(* CoDeSys 2.3.9.48 project: PLC_JBI.pro *)
(* Libraries: Util.lib 18.5.10 17:14:28, STANDARD.LIB 4.10.05 13:14:46, IECSFC.LIB 13.4.06 17:51:28, SYSLIBTIME.LIB 20.2.06 15:31:16, SYSTASKINFO.LIB 20.2.06 15:31:38, ANALYZATION.LIB 5.10.99 11:05:06, SYSLIBCALLBACK.LIB 20.2.06 15:31:08 *)

(* PLC configuration (modules and I/O channels)
Fast Counters [OWEN_ID531] node 0, in %IB0 out %QB0 {Visibility = No}
  di1_water AT %IW0.0 [WordInput] Fast counter 1
  di2_plast AT %IW0.1 [WordInput] Fast counter 2
AT %IB1.0 [ByteInput] 8 discrete inputs
AT %IB1.1 [ByteInput] 8 discrete inputs
Fast discrete outputs [OWEN_ID570] node 2, in %IB2 out %QB2 {SafeValueBool = FALSE; SafeValueBool = FALSE; SafeValueBool = FALSE; SafeValueBool = FALSE; Visibility = No}
  do1_comp_1 AT %QX2.0 [BitOutput] Fast discrete output 1
  do2_comp_2 AT %QX2.1 [BitOutput] Fast discrete output 2
  do3_comp_3 AT %QX2.2 [BitOutput] Fast discrete output 3
  do4_sem_raz AT %QX2.3 [BitOutput] Fast discrete output 4
Discrete outputs - 8 [ID131] node 3, in %IB3 out %QB3 {SafeValueByte = 0; Visibility = No; PinCount = 10}
  AT %QB3.0 [ByteOutput] 8 discrete outputs
Special input [ID103] node 4, in %IB4 out %QB4 {Filtrationtime = 1000; PinCount = 1; WatchDogPeriod = 400; PollPeriod = 3000; Visibility = No}
  AT %IX4.0 [BitInput] Special input
Special output [ID104] node 5, in %IB5 out %QB5 {Visibility = No; PinCount = 1}
  AT %QX5.0 [BitOutput] Special output
DCON (Master) [DCON_MASTER_ID452] node 6, in %IB6 out %QB6 {Visibility = No}
  AT %QW6.0 [WordOutput] Last error
  RS-485-2 [COM3_USART] node 0, in %IB6.0 out %QB6.0 {CommunicationSpeed = 11520; Parity = NO PARITY CHECK; BitLength = 8 bits; StopLength = One stop bit; InterfaceType = RS232; FrameOriented = ASCII; Timeout = 0; Visibility = No}
  Universal DCON device [ID2100] node 1, in %IB6.1 out %QB6.1 {ReqFormat = [15s]; GoodResponseFormat = !01[15s]; BadResponseFormat = ?; ServiceTimeout = 150; RequestType = By poll time; PeriodOfService = 100; Visibility = No}
    AT %QW6.1.0 [WordOutput] Status
cmd_plast AT %QB6.1.0.0 [StringOutput]
cntr_plast AT %IB6.1.1.0 [StringInput]
Universal DCON device [ID2100] node 2, in %IB6.2 out %QB6.2 {ReqFormat = [15s]; GoodResponseFormat = !02[15s]; BadResponseFormat = ?; ServiceTimeout = 150; RequestType = By poll time; PeriodOfService = 100; Visibility = No}
  AT %QW6.2.0 [WordOutput] Status
cmd_water AT %QB6.2.0.0 [StringOutput]
cntr_water AT %IB6.2.1.0 [StringInput]
Universal DCON device [ID2100] node 3, in %IB6.3 out %QB6.3 {ReqFormat = #01; GoodResponseFormat = >[8s]; BadResponseFormat = ?; ServiceTimeout = 150; RequestType = By poll time; PeriodOfService = 100; Visibility = No}
  AT %QW6.3.0 [WordOutput] Status
mVolt_sem AT %IB6.3.0.0 [StringInput]
Universal DCON device [ID2100] node 4, in %IB6.4 out %QB6.4 {ReqFormat = #02; GoodResponseFormat = >[8s]; BadResponseFormat = ?; ServiceTimeout = 150; RequestType = By poll time; PeriodOfService = 100; Visibility = No}
  AT %QW6.4.0 [WordOutput] Status
mVolt_sir AT %IB6.4.0.0 [StringInput]
AT %QW6.5.0 [WordOutput] Status
mVolt_wtr AT %IB6.5.0.0 [StringInput]
TCP [TCP_ID221] node 0, in %IB7.0.0 out %QB7.0.0 {RemotePort = 502; Visibility = No}
TCP [TCP_ID221] node 1, in %IB7.0.1 out %QB7.0.1 {RemotePort = 502; Visibility = No}
TCP [TCP_ID221] node 2, in %IB7.0.2 out %QB7.0.2 {RemotePort = 502; Visibility = No}
TCP [TCP_ID221] node 3, in %IB7.0.3 out %QB7.0.3 {RemotePort = 502; Visibility = No}
TCP [TCP_ID221] node 4, in %IB7.0.4 out %QB7.0.4 {RemotePort = 502; Visibility = No}
TCP [TCP_ID221] node 5, in %IB7.0.5 out %QB7.0.5 {RemotePort = 502; Visibility = No}
RS-232 [COM2_USART] node 6, in %IB7.0.6 out %QB7.0.6 {CommunicationSpeed = 11520; Parity = NO PARITY CHECK; BitLength = 8 bits; StopLength = One stop bit; InterfaceType = RS232; FrameOriented = RTU; Timeout = 10; Visibility = No}
Debug RS-232 [DEBUG_USART] node 7, in %IB7.0.7 out %QB7.0.7 {CommunicationSpeed = 11520; Parity = NO PARITY CHECK; BitLength = 8 bits; StopLength = One stop bit; InterfaceType = RS232; FrameOriented = RTU; Timeout = 10; Visibility = No}
8 bits [8Bit] node 1, in %IB7.1 out %QB7.1
  pc_mln_out1 AT %QB7.1.0 [ByteOutput] reg 0
8 bits [8Bit] node 2, in %IB7.2 out %QB7.2
  pc_mnl_out2 AT %QB7.2.0 [ByteOutput] reg 8
8 bits [8Bit] node 3, in %IB7.3 out %QB7.3
  pc_mnl_out3 AT %QB7.3.0 [ByteOutput] reg 16
8 bits [8Bit] node 4, in %IB7.4 out %QB7.4
  pc_mnl_in1 AT %QB7.4.0 [ByteOutput] reg 24
8 bits [8Bit] node 5, in %IB7.5 out %QB7.5
  pc_mnl_in2 AT %QB7.5.0 [ByteOutput] reg 32
8 bits [8Bit] node 6, in %IB7.6 out %QB7.6
  pc_mnl_in3 AT %QB7.6.0 [ByteOutput] reg 40
8 bits [8Bit] node 7, in %IB7.7 out %QB7.7
  AT %QB7.7.0 [ByteOutput] reg 48
8 bits [8Bit] node 8, in %IB7.8 out %QB7.8
  AT %QB7.8.0 [ByteOutput] reg 56
mb_local_sikl AT %QW7.9.0 [WordOutput]
mb_working_mode AT %QW7.10.0 [WordOutput]
mb_sikl AT %QW7.11.0 [WordOutput]
mb_tmr_conv AT %QW7.12.0 [WordOutput]
mb_tmr_comp1 AT %QW7.13.0 [WordOutput]
mb_tmr_comp2 AT %QW7.14.0 [WordOutput]
mb_tmr_comp3 AT %QW7.15.0 [WordOutput]
mb_tmr_mixer_bef AT %QW7.16.0 [WordOutput]
mb_tmr_shnk1 AT %QW7.17.0 [WordOutput]
mb_tmr_shnk2 AT %QW7.18.0 [WordOutput]
mb_tmr_water AT %QW7.19.0 [WordOutput]
mb_tmr_plast AT %QW7.20.0 [WordOutput]
mb_tmr_sem_bef AT %QW7.21.0 [WordOutput]
mb_tmr_bet AT %QW7.22.0 [WordOutput]
mb_tmr_skip_up AT %QW7.23.0 [WordOutput]
mb_tmr_skip_dwn AT %QW7.24.0 [WordOutput]
mb_tmr_skip_wait AT %QW7.25.0 [WordOutput]
mb_selct_shnk AT %QW7.26.0 [WordOutput]
mb_time_ET AT %QW7.27.0 [WordOutput]
AT %QW7.28.0 [WordOutput]
mb_weight_sem AT %QD7.29.0 [FloatOutput]
mb_weight_sir AT %QD7.30.0 [FloatOutput]
mb_weight_water AT %QD7.31.0 [FloatOutput]
mb_weight_plast AT %QD7.32.0 [FloatOutput]
mb_weight_sem_otkl AT %QD7.33.0 [FloatOutput]
mb_weight_sir_otkl AT %QD7.34.0 [FloatOutput]
mb_per_compo_1 AT %QD7.35.0 [FloatOutput]
mb_per_compo_2 AT %QD7.36.0 [FloatOutput]
mb_per_compo_3 AT %QD7.37.0 [FloatOutput]
mb_per_compo_total AT %QD7.38.0 [FloatOutput]
mb_tara_wht_sir AT %QD7.39.0 [FloatOutput]
mb_tara_wht_sem AT %QD7.40.0 [FloatOutput]
mb_weight_sem_zdn AT %QD7.41.0 [FloatOutput]
mb_weight_wtr_zdn AT %QD7.42.0 [FloatOutput]
mb_weight_comp1_zdn AT %QD7.43.0 [FloatOutput]
mb_weight_comp2_zdn AT %QD7.44.0 [FloatOutput]
mb_weight_comp3_zdn AT %QD7.45.0 [FloatOutput]
mb_weight_plast_zdn AT %QD7.46.0 [FloatOutput]
mb_tara_wht_water AT %QD7.47.0 [FloatOutput]
mb_tara_wht_plast AT %QD7.48.0 [FloatOutput]
AT %QD7.49.0 [FloatOutput]
AT %QD7.50.0 [FloatOutput]
mb_glob_sec AT %QW7.51.0 [WordOutput]
mb_mix_sec AT %QW7.52.0 [WordOutput]
mb_ERROR_code AT %QW7.53.0 [WordOutput]
AT %QW7.54.0 [WordOutput]
AT %QW7.55.0 [WordOutput]
AT %QW7.56.0 [WordOutput]
AT %QW7.57.0 [WordOutput]
AT %QW7.58.0 [WordOutput]
Button [ID003] node 8, in %IB8 out %QB8
  AT %IX8.0 [BitInput] Button Start/Stop
ModBus (Master) [MODBUS_MASTER_ID450] node 9, in %IB9 out %QB9 {Visibility = No}
  AT %QD9.0 [DWordOutput] Last address
  AT %QW9.1 [WordOutput] Last error
  RS-485-1 [COM1_USART] node 0, in %IB9.0 out %QB9.0 {CommunicationSpeed = 11520; Parity = NO PARITY CHECK; BitLength = 8 bits; StopLength = One stop bit; InterfaceType = RS485; FrameOriented = ASCII; Timeout = 0; Visibility = No}
AT %QB9.1.0 [ComChannel] Command (0xff - Start)
mdvv1_in AT %IW9.1.0.0 [WordInput]
mdvv1_out AT %QW9.1.1.0 [WordOutput]
AT %QB9.2.0 [ComChannel] Command (0xff - Start)
mdvv2_in AT %IW9.2.0.0 [WordInput]
mdvv2_out AT %QW9.2.1.0 [WordOutput]
*)

(* Global variable list: Global_Variables *)
VAR_GLOBAL
	klapON : BOOL;
	skipReady : BOOL;
	componentsREADY : BOOL;
	mixerNoREADY : BOOL;
	count_sir: BYTE;
	wtrimpl, plastimp : DWORD;
	allow_comp_1, allow_comp_2, allow_comp_3  : BOOL;
	allow_sem, allow_water, allow_plast  : BOOL;
	comp1 : compozits;
	comp2 : compozits;
	comp3 : compozits;
	mixer : mixers;
	skip : telejka;
	con : conveyr;
	sem : sements;
	wtr : water;
	plst : plastfikator;
	dreyf_sem : REAL;
	dreyf_sir : REAL;
	dreyf_wtr : REAL;
	(*********************)
	blinker : BLINK;
	cnt : CTU;
	cnt2 : CTU;
	cnt3 : CTU;
	GLOBT : DWORD;
	noERROR : BOOL ;
	(********************)
	kweight_sem : REAL;
	kweight_sir : REAL;
	kweight_wtr : REAL;
	kweight_plast : REAL;
END_VAR

(* Data type *)
TYPE compozits :
STRUCT
	ingroup : BOOL;
	zadan : REAL;
	run : BOOL;
	alarm : BOOL;
	status : BOOL;
	ready : BOOL := TRUE;
	allow : BOOL;
	vaqt1 : WORD;
	vaqt2 : WORD;
	sikl : WORD;
END_STRUCT
END_TYPE

(* Data type *)
TYPE conveyr :
STRUCT
	ready : BOOL := TRUE;
	run : BOOL;
	weight : REAL;
	tsikl : BOOL := TRUE;
	status : BOOL;
	tmr : TON;
	tmr_t : TIME;
	vaqt1 : WORD;
	vaqt2 : WORD;
	sikl : WORD;
END_STRUCT
END_TYPE

(* Data type *)
TYPE mixers :
STRUCT
	ready : BOOL;
	status : BOOL;
	open_cmd : BOOL;
	close_cmd : BOOL;
	lside: BOOL;
	rside : BOOL;
	open_sts : BOOL;
	close_sts : BOOL;
	vaqt1 : WORD;
	vaqt2 : WORD;
	sikl : WORD;

END_STRUCT
END_TYPE

(* Data type *)
TYPE plastfikator :
STRUCT
	run : BOOL;
	status : BOOL;
	zadan : REAL;
	ready : BOOL;
	level : REAL;
	enab : BOOL;
	vaqt1 : WORD;
	vaqt2 : WORD;
	sikl : WORD;
END_STRUCT
END_TYPE

(* Data type *)
TYPE sements :
STRUCT
	zadan : REAL;
	status : BOOL;
	ready : BOOL;
	run : BOOL;
	klapOPEN : BOOL;
	klapCLOSE : BOOL;
	vibr_cmd : BOOL;
	weight : REAL;
	dweight : REAL;
	open_cmd : BOOL;
	vaqt1 : WORD;
	vaqt2 : WORD;
	vaqt3 : WORD;
	vaqt4 : WORD;
	sikl : WORD;
END_STRUCT
END_TYPE

(* Data type *)
TYPE telejka :
STRUCT
	on_up : BOOL;
	on_down : BOOL;
	mov_up : BOOL;
	mov_dwn : BOOL;
	cmd_up : BOOL;
	cmd_dwn :BOOL;
	pause : BOOL;
	ready : BOOL;
	vaqt1 : WORD;
	vaqt2 : WORD;
	vaqt3 : WORD;
	vaqt4 : WORD;
	vaqt5 : WORD;
	sikl : WORD;
END_STRUCT
END_TYPE

(* Data type *)
TYPE water :
STRUCT
	run : BOOL;
	status : BOOL;
	zadan : REAL;
	ready : BOOL;
	level : REAL;
	enab : BOOL;
	vaqt1 : WORD;
	vaqt2 : WORD;
	sikl : WORD;
	unload : BOOL;
END_STRUCT
END_TYPE

(* POU PLC_PRG, ST *)
PROGRAM PLC_PRG
VAR
	tonMode : TON;
	tonVaqt : WORD := 300;
	tonReset : BOOL;
END_VAR
translate();
sikl_count();

IF 	(di18_sts_mnl = FALSE) THEN
		mb_cmd_start := FALSE;
		do6SkipStop := FALSE;
		mixerNoREADY := FALSE;
		(* mb_working_mode := 1;
		skip.cmd_up := FALSE;
		skip.cmd_dwn := FALSE;
		comp1.run := FALSE;
		comp2.run := FALSE;
		comp3.run := FALSE;
		con.run := FALSE;
		sem.run := FALSE;
		sem.open_cmd := FALSE;
		wtr.run := FALSE;
		plst.run := FALSE;

		cnt(reset := TRUE);
		cnt2(reset := TRUE);
		cnt3(reset := TRUE);
		componentsREADY := FALSE; *)
END_IF;
(*
IF 	(di18_sts_mnl = TRUE) AND
	(mb_cmd_start = TRUE) THEN
		(*mb_working_mode:= 0;*)
		cnt(reset := FALSE);
		cnt2(reset := FALSE);
		cnt3(reset := FALSE);
END_IF;
*)
mb_ERROR := (mb_ERROR_code <> 0);

CASE mb_working_mode OF
	0 : auto_half();
	1 : manual();
	2 : tara();
END_CASE;
IF mb_working_mode <> 2 THEN
	mb_working_mode := BOOL_TO_INT(NOT di18_sts_mnl);
END_IF;
tonMode(IN := (mb_working_mode = 2), PT := T#1s * tonVaqt);
IF (tonMode.Q = TRUE) THEN
	mb_working_mode := 1;
END_IF;

(*
IF 	(mb_working_mode < 0) OR
	(mb_working_mode > 2) THEN
		mb_working_mode := 1;
END_IF;
*)
END_PROGRAM

(* POU translate, ST *)
PROGRAM translate
VAR
	a: BOOL;
	tempimpw, tempimpp  : WORD;
	ftrig: F_TRIG;
	fltTON :TON;
	fltBool : BOOL;
	fltVaqt : WORD := 1000;
	t1, t2, t3 : REAL;
	suv : REAL;
	sumSuv : REAL;
	N : INT := 1;
	wtrOtkl : REAL := 15;
END_VAR
(*do5_water_klap := mb_cmd_wtr;
do9_plast_klap := mb_cmd_plst;*)
(*================== MDVV 1 OUT ==============================*)
mdvv1_out.0 := mb_cmd_raz_bet_opn ;
mdvv1_out.1 := mb_cmd_raz_bet_cls;
mdvv1_out.2 := mb_cmd_conveyr;
mdvv1_out.3 := mb_cmd_skip_dwn;
mdvv1_out.4 := mb_cmd_skip_up;
mdvv1_out.5 := mb_cmd_shnk1;
mdvv1_out.6 := mb_cmd_shnk2;
mdvv1_out.7 := mb_cmd_vibr;
(*==================================== MDVV 1 OUT ========================================*)
(*========================================================================================*)
mb_sts_comp_1 := di13_sts_comp_1;
mb_sts_comp_2 := di14_sts_comp_2;
mb_sts_comp_3 := di15_sts_comp_3;
mb_sts_water := di16_sts_water;
(*========================================================================================*)
(*========================================================================================*)
(*========================================================================================*)
(*=============================mdvv 1 in==================================================*)
mb_sts_mixer := mdvv1_in.0;
mb_sts_shnk_1 := mdvv1_in.1;
mb_sts_shnk_2 := mdvv1_in.2;
mb_sts_raz_betn_lf := mdvv1_in.3;
mb_sts_raz_betn_ri := NOT mdvv1_in.3;
mb_sts_vibrat := mdvv1_in.4;

mb_sts_conveyr := mdvv1_in.5;
mb_sts_plast := mdvv1_in.7;
mb_sts_kompr := mdvv1_in.6;
mb_sts_faza := mdvv1_in.8;
mb_sts_alrm_conveyr := mdvv1_in.9;
mb_sts_skp_move_dwn := mdvv1_in.10;
mb_sts_skp_move_up := mdvv1_in.11;
(*=========================mdvv 1 in ================================*)
(*===================================================================*)
(*==========================mdvv in 2 ===============================*)
(*==========================mdvv in 2 ===============================*)

mb_sts_skip_dwn     :=  NOT mdvv2_in.0;
mb_sts_skip_alrm_up := mdvv2_in.1;
mb_sts_skip_up      :=  NOT mdvv2_in.2;

mb_sts_mix_lf_opn   := mdvv2_in.3 AND mdvv2_in.4;(* mdvv2_in.3 - QS10- chap tomon ochiq    *************         mdvv2_in.4 - QS11 chap tomon yopiq*)
mb_sts_mix_ri_opn 	:= mdvv2_in.5 AND mdvv2_in.6;
mb_sts_raz_sem 		:= mdvv2_in.7 AND mdvv2_in.8;
mb_sts_telejka 		:= mdvv2_in.9;
mb_sts_skip_pause   := mdvv2_in.10;
mb_sts_skip_alrm_dwn := mdvv2_in.11;
(*==========================mdvv in 2 ===============================*)
(*==========================mdvv in 2 ===============================*)
(*================== PLC OUT ==============================*)

(*================== PLC OUT ==============================*)
(*================== MDVV 1 OUT ==============================*)
(*================== MDVV 1 OUT ==============================*)

(*============= MDVV 2 in ==============================*)
(*============= MDVV 2 in ==============================*)

(*============= MDVV 2 in ==============================*)
(*============= MDVV 2 in ==============================*)
fltTON(IN := fltBool, PT :=  T#1ms * fltVaqt);

mb_weight_sem := (STRING_TO_REAL(mVolt_sem) - dreyf_sem) * kweight_sem ;
mb_weight_sir := REAL_TO_INT((STRING_TO_REAL(mVolt_sir) - dreyf_sir) * kweight_sir); 
mb_weight_water := (STRING_TO_REAL(mVolt_wtr) - dreyf_wtr)* kweight_wtr;

(*
IF (fltTON.Q = TRUE) THEN
	mb_weight_water := suv;
	N:= 1;
ELSE
	sumSuv := (sumSuv + suv) / N;
	N := N + 1;
END_IF;
fltBool := NOT fltTON.Q;
IF (mb_weight_water < wtrOtkl) THEN
	klapON := TRUE;
END_IF;

IF (mb_weight_water > mb_weight_wtr_zdn) THEN
	klapON := FALSE;
END_IF;
*)
(*
IF (mb_cmd_wtr_nol = TRUE)THEN
	cmd_water := '@02CE';
	mb_cmd_wtr_nol := FALSE;

END_IF;

IF (mb_cmd_plast_nol = TRUE)THEN
	cmd_plast := '@01CE';
	mb_cmd_plast_nol := FALSE;

END_IF;
*)
IF 	(skip.on_up = TRUE) OR
	(mb_cmd_wtr_nol = TRUE) AND
	((mb_weight_plast > 0) OR
	(mb_weight_water > 0)) THEN
	cmd_water := '@02CE';
	cmd_plast := '@01CE';
ELSE
	cmd_water := '@02RE';
	cmd_plast := '@01RE';
END_IF;
(*

IF	(skip.on_down = TRUE) AND
	(mb_weight_water > 0) THEN
		mb_cmd_wtr_nol := TRUE;
END_IF;
IF	(skip.on_down = TRUE) AND
	(mb_weight_plast > 0) THEN
		mb_cmd_plast_nol := TRUE;
END_IF;*)

(*==============================================*)
(*==============================================*)
(*mb_weight_water := STRING_TO_REAL(cntr_water) * kweight_wtr; *)(* suvni hisoblagichga yig'ib borish*)
mb_weight_plast := STRING_TO_REAL(cntr_plast) * kweight_plast; (* plastifikatorni hisoblagichga yig'ib borish*)

IF (mb_cmd_sem_nol = TRUE) THEN
	dreyf_sem := STRING_TO_REAL(mVolt_sem);  (*sementni dreyv nolini kiritish*)
	mb_cmd_sem_nol := FALSE;
END_IF;

IF (mb_cmd_wtr_nol = TRUE) THEN
	dreyf_wtr := STRING_TO_REAL(mVolt_wtr);  (*sementni dreyv nolini kiritish*)
	mb_cmd_wtr_nol := FALSE;
END_IF;

IF (mb_cmd_sir_nol = TRUE) THEN
	dreyf_sir := STRING_TO_REAL(mVolt_sir);
	mb_cmd_sir_nol := FALSE;
END_IF;
(*====================================================================================*)

(*====================================================================================*)
IF 	(dreyf_sem = 0) THEN
		dreyf_sem := 3.48;
END_IF;
IF 	(dreyf_sir = 0) THEN
		dreyf_sir := 12.87;
END_IF;

IF 	(dreyf_wtr = 0) THEN
		dreyf_wtr := 3.319;
END_IF;
(*====================================================================================*)

(*
IF (di18_sts_mnl = FALSE) THEN
	skip.cmd_dwn := FALSE;
	skip.cmd_up := FALSE;
	comp1.run := FALSE;
	comp2.run := FALSE;
	comp3.run := FALSE;
	wtr.run := FALSE;
	plst.run := FALSE;
END_IF; *)
cnf_translt();
compo_trnslt();
skip_trnslt();
mix_trnslt();
water_trnslt();
plast_trnslt();
pc_mln_out1;
sel_shnk();
END_PROGRAM
ACTION cnf_translt:
IF(kweight_plast = 0) THEN
	kweight_plast := 0.015;
END_IF;
IF(kweight_wtr = 0) THEN
	kweight_wtr := 103.7736;
END_IF;
IF(kweight_sem = 0) THEN
	kweight_sem := 45;
END_IF;
IF(kweight_sir = 0 OR kweight_sir > 306) THEN
	kweight_sir := 247;
END_IF;
END_ACTION
ACTION compo_trnslt:
(*======================================================*)
(*====================comp1==================================*)
comp1.ingroup := (mb_weight_comp1_zdn > 0) AND
				 (mb_cmd_start = TRUE) AND
				 (di18_sts_mnl = TRUE) AND
				 (mb_local_sikl <= mb_sikl);
comp1.status := mb_sts_comp_1;
(*do1_comp_1 := comp1.run;*)
comp1.zadan := mb_weight_comp1_zdn;
(*======================================================*)
(*=======================comp2===============================*)
comp2.ingroup := (mb_weight_comp2_zdn > 0) AND
				 (mb_cmd_start = TRUE) AND
				 (di18_sts_mnl = TRUE) AND
				 (mb_local_sikl <= mb_sikl);
comp2.status := mb_sts_comp_2;
(*do2_comp_2 := comp2.run; *)
comp2.zadan := mb_weight_comp2_zdn;
(*============================================================*)
(*=======================comp3===============================*)
comp3.ingroup := (mb_weight_comp3_zdn > 0) AND
				 (mb_cmd_start = TRUE) AND
				 (di18_sts_mnl = TRUE) AND
				 (mb_local_sikl <= mb_sikl);
comp3.status := mb_sts_comp_3;
(*do3_comp_3 := comp3.run;*)
comp3.zadan := mb_weight_comp3_zdn;
(*=============================================================*)
(*=======================conveyr===============================*)
mb_cmd_conveyr := con.run;
con.status := mb_sts_conveyr;
con.weight := mb_weight_sir;

(*=============================================================*)
(*=============================================================*)
END_ACTION
ACTION mix_trnslt:
(*====================================================================================*)
(*====================================================================================*)
sem.zadan := mb_weight_sem_zdn;
sem.weight := (STRING_TO_REAL(mVolt_sem) - dreyf_sem)* kweight_sem ;
sem.klapCLOSE := mdvv2_in.7;
sem.klapOPEN := mdvv2_in.8;
sem.status := mdvv1_in.1 OR mdvv1_in.2;
mdvv1_out.7 := sem.vibr_cmd;
do4_sem_raz := sem.open_cmd;
(*====================================================================================*)
(*====================================================================================*)
mixer.open_sts := (mdvv2_in.3 = TRUE) OR (mdvv2_in.5 = TRUE);
mixer.close_sts := (mdvv2_in.4 = TRUE) AND (mdvv2_in.6 = TRUE);
mixer.status := mdvv1_in.0;

(*
mdvv1_out.0 := mixer.open_cmd;
mdvv1_out.1 := mixer.close_cmd;
*)
mixer.lside := mdvv1_in.3;
mixer.rside := NOT mdvv1_in.3;

(*====================================================================================*)
(*====================================================================================*)



(*====================================================================================*)
(*====================================================================================*)
END_ACTION
ACTION plast_trnslt:
plst.level := STRING_TO_REAL(cntr_plast) * kweight_plast;
plst.zadan := mb_weight_plast_zdn;
do9_plast_klap := plst.run;
plst.status := di17_sts_plast;
END_ACTION
ACTION sel_shnk:
IF (mb_sel_shnk = TRUE) THEN
	mdvv1_out.5 := sem.run;
ELSE
	mdvv1_out.6 := sem.run;
END_IF;
END_ACTION
ACTION skip_trnslt:
mdvv1_out.3 := skip.cmd_dwn;
mdvv1_out.4 := skip.cmd_up;
skip.mov_dwn := mdvv1_in.10;
skip.mov_up := mdvv1_in.11;
skip.on_down := NOT mdvv2_in.0;
skip.on_up := NOT mdvv2_in.2;
skip.pause := mdvv2_in.9;
END_ACTION
ACTION water_trnslt:
wtr.level := STRING_TO_REAL(cntr_water) * kweight_wtr;
wtr.zadan := mb_weight_wtr_zdn;
(*do5_water_klap := wtr.run;*)
wtr.status := di16_sts_water;
END_ACTION

(* POU sikl_count, CFC *)
PROGRAM sikl_count
VAR
	och_yop: F_TRIG;
	tonCount: TON;
	vaqt : WORD := 5;
END_VAR
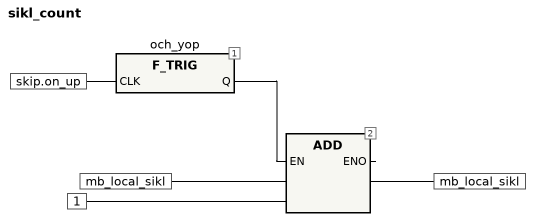
_CFC_ (* Continuous Function Chart, elements in execution order *)
#0 mb_local_sikl <= #2
#1 och_yop:F_TRIG(CLK: skip.on_up)
#2 ADD(EN: #1.Q, mb_local_sikl, 1)
_END_CFC_
END_PROGRAM

(* POU auto_half, ST *)
PROGRAM auto_half
VAR
END_VAR
mixerAdjust();
dozersAndConv();
sementAdjust();
waterAdjust();
skipAdjust();
END_PROGRAM

(* POU mixerAdjust, ST *)
PROGRAM mixerAdjust
VAR
	STEP : WORD := 0;
	ton1 : TON;
	ton2 : TON;
	ton1Time : TIME := T#10s;
	rtrig : R_TRIG;
	temp : BOOL;
END_VAR
IF (mixer.open_sts) THEN
	mixerNoREADY := TRUE;
END_IF;
ton1(IN := mixer.open_sts, PT := ton1Time);
mb_time_ET := TIME_TO_WORD(ton1.ET) / 1000;
rtrig(CLK := ton1.Q);
IF (rtrig.Q = TRUE) THEN
	temp := TRUE;
END_IF;
ton2(IN := mixer.close_sts = TRUE AND temp = TRUE, PT := T#5s);
IF (ton2.Q) THEN
	mixerNoREADY := FALSE;
	temp := FALSE;
END_IF;
END_PROGRAM

(* POU dozersAndConv, ST *)
PROGRAM dozersAndConv
VAR
	STEP : WORD := 0;
	run: BOOL;
	ton1 : TON;
	ton2 : TON;
	ton3 : TON;
	ton4 : TON;
	tpConv : TP;
	tpTimeConv : TIME := T#7s;
	waitTime : TIME := T#2s;
	waitTimeConv : TIME := T#1s;
	weightOtkl : REAL := 17;
END_VAR
run :=
	mb_cmd_start
	AND di18_sts_mnl;
CASE STEP OF
	0 :
		ton1(IN := mb_weight_sir + 10 >= mb_weight_comp1_zdn, PT := waitTime);
		IF (mb_weight_comp1_zdn > 0 AND mb_weight_sir + 10 < mb_weight_comp1_zdn) THEN
			do1_comp_1 := run;
			do2_comp_2 := FALSE;
			do3_comp_3 := FALSE;
		ELSE
			do1_comp_1 := FALSE;
			do2_comp_2 := FALSE;
			do3_comp_3 := FALSE;
			IF (ton1.Q = TRUE) THEN
				STEP := 1;
			END_IF;
		END_IF;
		IF ( di18_sts_mnl = FALSE) THEN
			STEP := 0;
		END_IF;
	1 :
		ton2(IN := mb_weight_sir + 10 >= mb_weight_comp1_zdn + mb_weight_comp2_zdn, PT := waitTime);
		IF (mb_weight_comp2_zdn > 0 AND mb_weight_sir + 10 < mb_weight_comp1_zdn + mb_weight_comp2_zdn) THEN
			do1_comp_1 := FALSE;
			do2_comp_2 := run;
			do3_comp_3 := FALSE;
		ELSE
			do1_comp_1 := FALSE;
			do2_comp_2 := FALSE;
			do3_comp_3 := FALSE;
			IF(ton2.Q = TRUE) THEN
				STEP := 2;
			END_IF;
		END_IF;
		IF ( di18_sts_mnl = FALSE) THEN
			STEP := 0;
		END_IF;
	2 :
		ton3(IN := mb_weight_sir + 10 >= mb_weight_comp1_zdn + mb_weight_comp2_zdn + mb_weight_comp3_zdn, PT := waitTime);
		IF (mb_weight_comp3_zdn > 0 AND mb_weight_sir + 10 < mb_weight_comp1_zdn + mb_weight_comp2_zdn + mb_weight_comp3_zdn) THEN
			do1_comp_1 := FALSE;
			do2_comp_2 := FALSE;
			do3_comp_3 := run;
		ELSE
			do1_comp_1 := FALSE;
			do2_comp_2 := FALSE;
			do3_comp_3 := FALSE;
			IF (ton3.Q = TRUE) THEN
				STEP := 3;
			END_IF;
		END_IF;
		IF ( di18_sts_mnl = FALSE) THEN
			STEP := 0;
		END_IF;
	3 :	tpConv(IN := mb_weight_sir <= weightOtkl , PT := tpTimeConv);
		ton4(IN := NOT con.run, PT := waitTimeConv);
		IF (do1_comp_1 = FALSE AND skip.on_down = TRUE
						AND do2_comp_2 = FALSE
						AND do3_comp_3 = FALSE
						AND (mb_weight_sir > weightOtkl
						OR tpConv.Q = TRUE)) THEN
			con.run := run;
			comp1.run := FALSE;
			comp2.run := FALSE;
			comp3.run := FALSE;
		ELSIF (mb_weight_sir <= weightOtkl OR NOT skip.on_down) THEN
			con.run := FALSE;
			IF (ton4.Q = TRUE) THEN
				STEP := 0;
			END_IF;
		END_IF;
		IF ( di18_sts_mnl = FALSE) THEN
			STEP := 0;
		END_IF;
END_CASE;
END_PROGRAM

(* POU sementAdjust, ST *)
PROGRAM sementAdjust
VAR
	STEP : WORD;
	run: BOOL;
	ton1 : TON;
	ton2 : TON;
	ton3 : TON;
	waitTime : TIME := T#3s;
	waitTimeThrow : TIME := T#8s;
	weight_sem_otkl: REAL := 30;
	ftrig : F_TRIG;
	temp : BOOL;
END_VAR
run :=
	di18_sts_mnl AND
	mb_cmd_start;
CASE STEP OF
	0 :
		ton1(IN := mb_weight_sem >= mb_weight_sem_zdn AND NOT do4_sem_raz, PT := waitTime);
		IF (mb_weight_sem < mb_weight_sem_zdn AND mb_weight_sem_zdn > 0 AND NOT do4_sem_raz) THEN
			sem.run := run;
		ELSE
			sem.run := FALSE;
			IF (ton1.Q = TRUE) THEN
				STEP := 1;
				sem.run := FALSE;
			END_IF;
		END_IF;
		IF ( di18_sts_mnl = FALSE) THEN
			STEP := 0;
		END_IF;
		temp := FALSE;
	1 :
		ftrig(CLK := skip.on_up);
		IF (ftrig.Q = TRUE) THEN
			temp := TRUE;
		END_IF;
		ton2(IN := temp, PT := waitTimeThrow);
		IF (mb_weight_sem > weight_sem_otkl AND ton2.Q = TRUE AND mixer.close_sts) THEN
			do4_sem_raz := run;
		ELSE
			IF (ton2.Q = TRUE) THEN
				STEP := 2;
			END_IF;
			do4_sem_raz := FALSE;
		END_IF;
		IF ( di18_sts_mnl = FALSE) THEN
			STEP := 0;
		END_IF;
	2 :
		ton3(IN := temp, PT := T#3s);
		IF ( di18_sts_mnl = FALSE) THEN
			STEP := 0;
		END_IF;
		temp := FALSE;
		STEP := 0;
END_CASE;
END_PROGRAM

(* POU waterAdjust, ST *)
PROGRAM waterAdjust
VAR
	STEP : WORD;
	run: BOOL;
	ton1 : TON;
	ton2 : TON;
	ftrig : F_TRIG;
	temp : BOOL;
	waitTime : TIME := T#10ms;
	waitTimeFill : TIME := T#7s;
	weightOtkl : REAL := 10;
END_VAR
run :=
	di18_sts_mnl AND
	mb_cmd_start;
ftrig(CLK := mixer.open_sts);
IF (ftrig.Q = TRUE) THEN
	temp := TRUE;
END_IF;
CASE STEP OF
	0 :
		ton1(IN := mb_weight_water + 5 >= mb_weight_wtr_zdn, PT := waitTime);
		IF (mb_weight_water < mb_weight_wtr_zdn AND mb_weight_wtr_zdn > 15) THEN
			do5_water_klap := run;
		ELSE
			do5_water_klap := FALSE;
			IF (ton1.Q = TRUE) THEN
				STEP := 1;
				temp := FALSE;
			END_IF;
		END_IF;
		IF ( di18_sts_mnl = FALSE) THEN
			STEP := 0;
		END_IF;
	1 :
		(*ton2(IN := mb_weight_water < weightOtkl AND mixer.open_sts, PT := waitTimeFill);*)
		ton2(IN := temp, PT := waitTimeFill);
		IF (ton2.Q = TRUE) THEN
			STEP := 0;
			temp := FALSE;
		END_IF;
		IF ( di18_sts_mnl = FALSE) THEN
			STEP := 0;
		END_IF;
END_CASE;
END_PROGRAM

(* POU skipAdjust, ST *)
PROGRAM skipAdjust
VAR
	STEP : WORD;
	run: BOOL;
	ftrig : F_TRIG;
	ftrigP : F_TRIG;
	temp : BOOL;
	ton0 : TON;
	ton1 : TON;
	tonPause : TON;
	timePause : TIME := T#30s;
	waitOnTopTime : TIME := T#5s;
	tempP : BOOL;
END_VAR
run :=
	di18_sts_mnl AND
	mb_cmd_start;
tonPause(IN :=
	NOT skip.on_down AND
	NOT skip.on_up, PT := timePause);
CASE STEP OF
	0 :	ftrig(CLK := con.run);
		tempP := FALSE;
		do6SkipStop := FALSE;
		skip.cmd_dwn := FALSE;
		skip.cmd_up := FALSE;
		IF (ftrig.Q = TRUE) THEN
			temp := TRUE;
		END_IF;
		ton0(IN := temp, PT := T#9s);
		IF (ton0.Q = TRUE) THEN
			temp := FALSE;
			STEP := 1;
		END_IF;
		IF ( di18_sts_mnl = FALSE) THEN
			STEP := 0;
		END_IF;
	1 :
		skip.cmd_up := run;
		skip.cmd_dwn := FALSE;
		IF (skip.on_down = FALSE) THEN
			STEP := 2;
			skip.cmd_up := FALSE;
		END_IF;
		IF (di18_sts_mnl = FALSE) THEN
			STEP := 0;
		END_IF;
	2 :
		IF ((tonPause.Q = TRUE OR skip.pause = TRUE) AND (do6SkipStop = FALSE)) THEN
			do6SkipStop := TRUE;
			skip.cmd_dwn := FALSE;
			skip.cmd_up := FALSE;
		END_IF;
		IF (mixerNoREADY = FALSE AND
			mb_weight_sem >= mb_weight_sem_zdn AND
			mb_weight_water >= mb_weight_wtr_zdn) THEN
			do6SkipStop := FALSE;
			STEP := 3;
			skip.cmd_up := FALSE;
		END_IF;
		IF ( di18_sts_mnl = FALSE) THEN
			STEP := 0;
		END_IF;
	3 :
		ton1(IN := skip.on_up, PT := waitOnTopTime);
		IF (skip.on_up = FALSE) THEN
			skip.cmd_dwn := FALSE;
			skip.cmd_up := run;
			do6SkipStop := mixerNoREADY;
		ELSE
			skip.cmd_dwn := FALSE;
			skip.cmd_up := FALSE;
		END_IF;
		IF (ton1.Q = TRUE) THEN
			STEP := 4;
			mixerNoREADY := TRUE;
		END_IF;
		IF ( di18_sts_mnl = FALSE) THEN
			STEP := 0;
		END_IF;
	4 :
		IF (skip.on_up = TRUE) THEN
			skip.cmd_dwn := run;
			skip.cmd_up := FALSE;
		ELSE
			skip.cmd_dwn := FALSE;
			skip.cmd_up := FALSE;
		END_IF;
		IF (skip.on_down = TRUE) THEN
			STEP := 0;
			skip.cmd_dwn := FALSE;
			skip.cmd_up := FALSE;
			tempP := FALSE;
		END_IF;
		IF ( di18_sts_mnl = FALSE) THEN
			STEP := 0;
		END_IF;
END_CASE;
IF (skip.on_down = TRUE AND run = FALSE) THEN
	STEP := 0;
	do6SkipStop := FALSE;
	skip.cmd_dwn := FALSE;
	skip.cmd_up := FALSE;
END_IF;
END_PROGRAM

(* POU manual, ST *)
PROGRAM manual
VAR
	increm : BOOL;
END_VAR
IF (di18_sts_mnl = FALSE)  THEN
	manual_ld();
END_IF;
mnl_yuk_chk();
IF 	(mb_sts_skip_up = TRUE AND
	 do4_sem_raz = TRUE ) THEN
		IF (increm = TRUE) THEN
			mb_weight_water := 0;
			mb_weight_plast := 0;
			increm := FALSE;
		END_IF;
END_IF;
IF 	(mb_sts_mix_lf_opn = TRUE OR
	 mb_sts_mix_ri_opn = TRUE) THEN
		increm := TRUE;
END_IF;
END_PROGRAM

(* POU manual_ld, LD *)
PROGRAM manual_ld
VAR
	b1: BOOL;
	s1: BOOL;
	counter : CTU;
	btrg: R_TRIG;
	sr1: SR;
	enb : BOOL;
	ton1: TP;

	btrg2: F_TRIG;
	rst : BOOL;
	rvrs: BOOL;
	ctt: CTU;
END_VAR
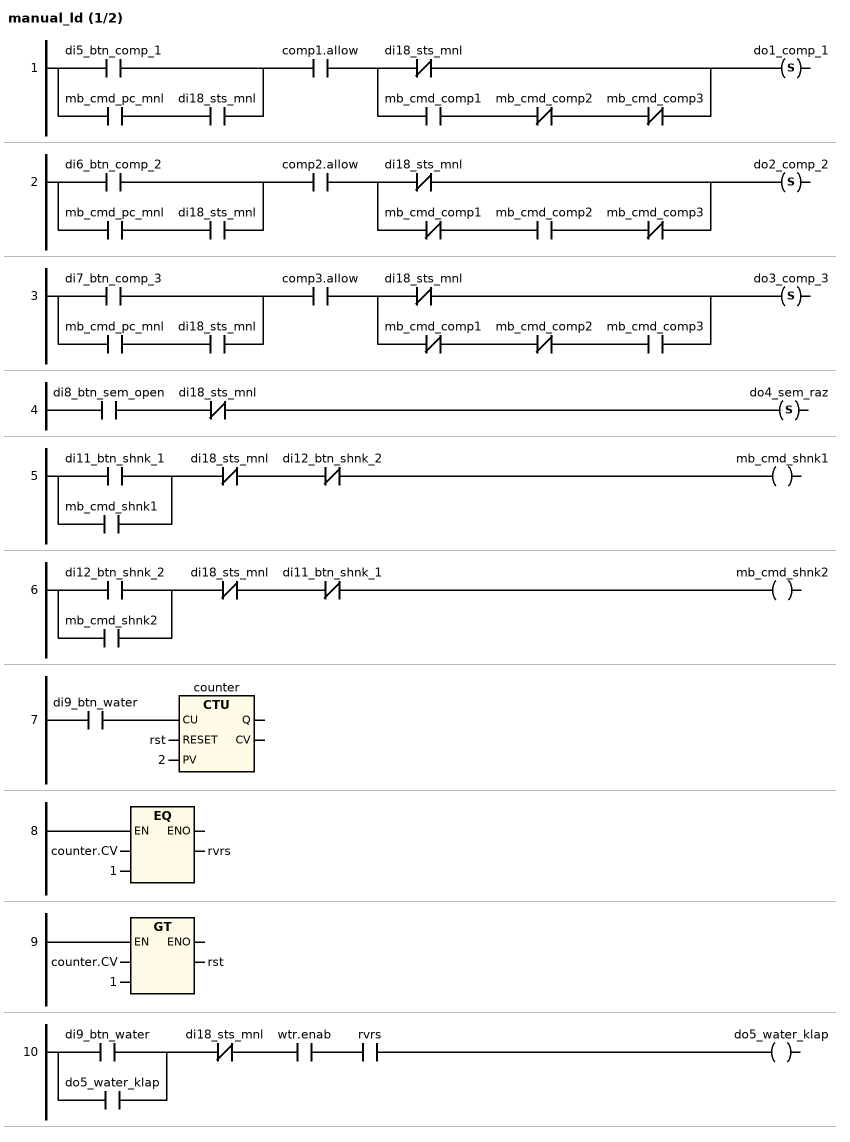
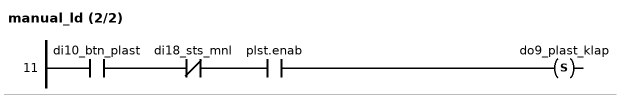
_LD_ (* Ladder Diagram *)
NETWORK 1
	{ [di5_btn_comp_1] | [mb_cmd_pc_mnl] - [di18_sts_mnl] } - [comp1.allow] - { [/di18_sts_mnl] | [mb_cmd_comp1] - [/mb_cmd_comp2] - [/mb_cmd_comp3] } --- (S do1_comp_1)
NETWORK 2
	{ [di6_btn_comp_2] | [mb_cmd_pc_mnl] - [di18_sts_mnl] } - [comp2.allow] - { [/di18_sts_mnl] | [/mb_cmd_comp1] - [mb_cmd_comp2] - [/mb_cmd_comp3] } --- (S do2_comp_2)
NETWORK 3
	{ [di7_btn_comp_3] | [mb_cmd_pc_mnl] - [di18_sts_mnl] } - [comp3.allow] - { [/di18_sts_mnl] | [/mb_cmd_comp1] - [/mb_cmd_comp2] - [mb_cmd_comp3] } --- (S do3_comp_3)
NETWORK 4
	[di8_btn_sem_open] - [/di18_sts_mnl] --- (S do4_sem_raz)
NETWORK 5
	{ [di11_btn_shnk_1] | [mb_cmd_shnk1] } - [/di18_sts_mnl] - [/di12_btn_shnk_2] --- (mb_cmd_shnk1)
NETWORK 6
	{ [di12_btn_shnk_2] | [mb_cmd_shnk2] } - [/di18_sts_mnl] - [/di11_btn_shnk_1] --- (mb_cmd_shnk2)
NETWORK 7
	[di9_btn_water] - counter:CTU(CU: *, RESET: rst, PV: 2)
NETWORK 8
	*
		EN --- EQ(counter.CV, 1) => rvrs
NETWORK 9
	*
		EN --- GT(counter.CV, 1) => rst
NETWORK 10
	{ [di9_btn_water] | [do5_water_klap] } - [/di18_sts_mnl] - [wtr.enab] - [rvrs] --- (do5_water_klap)
NETWORK 11
	[di10_btn_plast] - [/di18_sts_mnl] - [plst.enab] --- (S do9_plast_klap)
_END_LD_
(* the same logic as Structured Text *)
(* Network 1 *)
IF (di5_btn_comp_1 OR mb_cmd_pc_mnl AND di18_sts_mnl) AND comp1.allow AND (NOT di18_sts_mnl OR mb_cmd_comp1 AND NOT mb_cmd_comp2 AND NOT mb_cmd_comp3) THEN do1_comp_1 := TRUE; END_IF;
(* Network 2 *)
IF (di6_btn_comp_2 OR mb_cmd_pc_mnl AND di18_sts_mnl) AND comp2.allow AND (NOT di18_sts_mnl OR NOT mb_cmd_comp1 AND mb_cmd_comp2 AND NOT mb_cmd_comp3) THEN do2_comp_2 := TRUE; END_IF;
(* Network 3 *)
IF (di7_btn_comp_3 OR mb_cmd_pc_mnl AND di18_sts_mnl) AND comp3.allow AND (NOT di18_sts_mnl OR NOT mb_cmd_comp1 AND NOT mb_cmd_comp2 AND mb_cmd_comp3) THEN do3_comp_3 := TRUE; END_IF;
(* Network 4 *)
IF di8_btn_sem_open AND NOT di18_sts_mnl THEN do4_sem_raz := TRUE; END_IF;
(* Network 5 *)
mb_cmd_shnk1 := (di11_btn_shnk_1 OR mb_cmd_shnk1) AND NOT di18_sts_mnl AND NOT di12_btn_shnk_2;
(* Network 6 *)
mb_cmd_shnk2 := (di12_btn_shnk_2 OR mb_cmd_shnk2) AND NOT di18_sts_mnl AND NOT di11_btn_shnk_1;
(* Network 7 *)
counter(CU := di9_btn_water, RESET := rst, PV := 2);
(* Network 8 *)
rvrs := counter.CV = 1;
(* Network 9 *)
rst := counter.CV > 1;
(* Network 10 *)
do5_water_klap := (di9_btn_water OR do5_water_klap) AND NOT di18_sts_mnl AND wtr.enab AND rvrs;
(* Network 11 *)
IF di10_btn_plast AND NOT di18_sts_mnl AND plst.enab THEN do9_plast_klap := TRUE; END_IF;
END_PROGRAM

(* POU mnl_yuk_chk, ST *)
PROGRAM mnl_yuk_chk
VAR
	tmp_real : REAL;
	tmp_bool : BOOL;
	otkl1 : REAL := 10;
	otkl2 : REAL := 10;
	otkl3 : REAL := 10;
	cntW: CTU;
END_VAR
(*+++++++++++++++++++++++++++++++++++++++++++++++++++++++++++++++++++
IF (count_sir = 0) THEN
	allow_comp_1 := TRUE;
ELSE
	allow_comp_1 := FALSE;
END_IF;*)


IF ((di5_btn_comp_1 = TRUE) OR (mb_cmd_comp1 =TRUE) AND (mb_cmd_pc_mnl = TRUE)) AND (tmp_bool = TRUE) THEN
	tmp_real := mb_weight_sir;
	tmp_bool := FALSE;
END_IF;
IF	(mb_weight_comp1_zdn - otkl1  <= mb_weight_sir) OR
	(mb_sts_conveyr = TRUE)(* + tmp_real*) THEN
		do1_comp_1 := FALSE;
		tmp_bool := TRUE;
		count_sir := 1;
END_IF;
IF (di6_btn_comp_2 = TRUE OR di7_btn_comp_3 = TRUE AND di18_sts_mnl = FALSE) OR (mb_cmd_comp1 = FALSE AND di18_sts_mnl = TRUE) THEN
	do1_comp_1 := FALSE;
END_IF;
(*+++++++++++++++++++++++++++++++++++++++++++++++++++++++++++++++++++*)

(*+++++++++++++++++++++++++++++++++++++++++++++++++++++++++++++++++++
IF (count_sir = 1) THEN
	allow_comp_2 := TRUE;
ELSE
	allow_comp_2 := FALSE;
END_IF;*)
IF (di6_btn_comp_2 = TRUE) AND (tmp_bool = TRUE) OR ((mb_cmd_comp2 =TRUE) AND (mb_cmd_pc_mnl = TRUE)) THEN
	tmp_real := mb_weight_sir;
	tmp_bool := FALSE;
END_IF;
IF 	((mb_weight_comp2_zdn + mb_weight_comp1_zdn) - otkl2 < mb_weight_sir) OR
	(mb_sts_conveyr = TRUE)(* + tmp_real*) THEN
	do2_comp_2 := FALSE;
	tmp_bool := TRUE;
	count_sir := 2;
END_IF;
IF (di5_btn_comp_1 OR di7_btn_comp_3)OR((mb_cmd_comp2 = FALSE) AND (mb_cmd_pc_mnl = TRUE)) THEN
	do2_comp_2 := FALSE;
END_IF;
(*+++++++++++++++++++++++++++++++++++++++++++++++++++++++++++++++++++*)

(*+++++++++++++++++++++++++++++++++++++++++++++++++++++++++++++++++++
IF (count_sir = 2) THEN
	allow_comp_3 := TRUE;
ELSE
	allow_comp_3 := FALSE;
END_IF;*)
IF (di7_btn_comp_3 = TRUE) AND (tmp_bool = TRUE) OR ((mb_cmd_comp3 =TRUE) AND (mb_cmd_pc_mnl = TRUE)) THEN
	tmp_real := mb_weight_sir;
	tmp_bool := FALSE;
END_IF;
IF ((mb_weight_comp1_zdn + mb_weight_comp2_zdn + mb_weight_comp3_zdn) - otkl3 < mb_weight_sir)(* + tmp_real*)
	OR 	(mb_sts_conveyr = TRUE) THEN
	do3_comp_3 := FALSE;
	tmp_bool := TRUE;
	count_sir := 0;
END_IF;
IF (di5_btn_comp_1 OR di6_btn_comp_2)OR ((mb_cmd_comp3 =TRUE) AND (mb_cmd_pc_mnl = TRUE)) THEN
	do3_comp_3 := FALSE;
END_IF;
(*+++++++++++++++++++++++++++++++++++++++++++++++++++++++++++++++++++*)
(*+++++++++++++++++++++++++++++++++++++++++++++++++++++++++++++++++++*)
IF 	(mb_weight_sem >= mb_weight_sem_zdn) THEN
		mb_cmd_shnk1 := FALSE;
		mb_cmd_shnk2 := FALSE;
END_IF;
(*+++++++++++++++++++++++++++++++++++++++++++++++++++++++++++++++++++*)
(*+++++++++++++++++++++++++++++++++++++++++++++++++++++++++++++++++++*)
IF 	(mb_weight_water + 4 >= mb_weight_wtr_zdn) OR
	(mb_weight_wtr_zdn <= 0) THEN
		wtr.enab := FALSE;
		do5_water_klap := FALSE;
ELSE
		wtr.enab := TRUE;
END_IF;
(*+++++++++++++++++++++++++++++++++++++++++++++++++++++++++++++++++++*)
(*+++++++++++++++++++++++++++++++++++++++++++++++++++++++++++++++++++*)
IF  (mb_weight_plast >= mb_weight_plast_zdn) OR
	(mb_weight_plast_zdn <= 0 ) THEN
		do9_plast_klap := FALSE;
		plst.enab := FALSE;
ELSE
		plst.enab := TRUE;
END_IF
IF 	(mb_cmd_shnk1 = TRUE) OR
	(mb_cmd_shnk2 = TRUE) OR
	(do5_water_klap = TRUE) OR
	(do9_plast_klap= TRUE) THEN
		do4_sem_raz := FALSE;
END_IF;

(*+++++++++++++++++++++++++++++++++++++++++++++++++++++++++++++++++++*)
(*+++++++++++++++++++++++++++++++++++++++++++++++++++++++++++++++++++*)
IF(di18_sts_mnl = TRUE) THEN
	mb_cmd_comp1 := FALSE;
	mb_cmd_comp2 := FALSE;
	mb_cmd_comp3 := FALSE;
	do1_comp_1 := FALSE;
	do2_comp_2 := FALSE;
	do3_comp_3 := FALSE;
	mb_cmd_shnk1 := FALSE;
	mb_cmd_shnk2 := FALSE;
END_IF;
(*+++++++++++++++++++++++++++++++++++++++++++++++++++++++++++++++++++*)
selct_comp();
END_PROGRAM

(* POU selct_comp, ST *)
PROGRAM selct_comp
VAR
END_VAR
IF 	(mb_weight_sir_otkl >= mb_weight_sir) AND
	(mb_weight_sir_otkl + mb_weight_sir <= mb_weight_comp1_zdn) THEN
		comp1.allow := TRUE;
		comp2.allow := FALSE;
		comp3.allow := FALSE;
END_IF;
IF 	(mb_weight_sir_otkl + mb_weight_sir >= mb_weight_comp1_zdn) AND
	(mb_weight_sir_otkl + mb_weight_sir <= mb_weight_comp2_zdn + mb_weight_comp1_zdn) THEN
		comp1.allow := FALSE;
		comp2.allow := TRUE;
		comp3.allow := FALSE;
END_IF;
IF 	(mb_weight_sir_otkl + mb_weight_sir >= mb_weight_comp2_zdn + mb_weight_comp1_zdn) AND
	(mb_weight_sir_otkl + mb_weight_sir <= mb_weight_comp3_zdn + mb_weight_comp2_zdn + mb_weight_comp1_zdn) THEN
		comp1.allow := FALSE;
		comp2.allow := FALSE;
		comp3.allow := TRUE;
END_IF;
END_PROGRAM

(* POU tara, ST *)
PROGRAM tara
VAR
END_VAR
IF(mb_cmd_kwht_sem = TRUE) THEN
	IF (STRING_TO_REAL(mVolt_sir) > 0) THEN
		kweight_sem := mb_tara_wht_sem / (STRING_TO_REAL(mVolt_sem) - dreyf_sem);
	ELSE
		kweight_sem := 45.45454;
	END_IF;
	mb_cmd_kwht_sem := FALSE;
END_IF;
IF(mb_cmd_kwht_sir = TRUE) THEN
	IF (STRING_TO_REAL(mVolt_sir) > 0) THEN
		kweight_sir := mb_tara_wht_sir / (STRING_TO_REAL(mVolt_sir) - dreyf_sir);
	ELSE
		kweight_sir := 247.0587;
	END_IF;
	mb_cmd_kwht_sir := FALSE;
END_IF;
IF (mb_cmd_kwht_water = TRUE) THEN
	IF	(STRING_TO_REAL(mVolt_wtr) > 0) THEN
			kweight_wtr := mb_tara_wht_water / (STRING_TO_REAL(mVolt_wtr) - dreyf_wtr);
	ELSE
			kweight_wtr := 104.4776;
	END_IF;
	mb_cmd_kwht_water := FALSE;
END_IF;
IF (mb_cmd_kwht_plast = TRUE) THEN
	IF 	(STRING_TO_REAL(cntr_plast) > 0) THEN
			kweight_plast := mb_tara_wht_plast / STRING_TO_REAL(cntr_plast);
	ELSE
			kweight_plast := mb_tara_wht_plast;
	END_IF;
	mb_cmd_kwht_plast := FALSE;
END_IF;
END_PROGRAM

(* POU sementAdjust_1, ST *)
PROGRAM sementAdjust_1
VAR
	STEP : WORD;
	run: BOOL;

	ton1 : TON;
	ton2 : TON;
	ton3 : TON;
	waitTime : TIME := T#3s;
	waitTimeThrow : TIME := T#5s;
	weight_sem_otkl: REAL := 10;
	ftrig : F_TRIG;
	temp : BOOL;
END_VAR
run := di18_sts_mnl AND mb_cmd_start;


CASE STEP OF
	0 :
		ton1(IN := mb_weight_sem >= mb_weight_sem_zdn AND NOT sem.open_cmd, PT := waitTime);
		IF (mb_weight_sem < mb_weight_sem_zdn AND mb_weight_sem_zdn > 0 AND NOT do4_sem_raz) THEN
			sem.run := run;
		ELSE
			sem.run := FALSE;
			IF (ton1.Q = TRUE) THEN
				STEP := 1;
			END_IF;
		END_IF;
	1 :
		ton1(IN := skip.on_up, PT := waitTimeThrow);
		IF (ton1.Q = TRUE) THEN
			STEP := 2;
		END_IF;
	2 : ton2(IN := mb_weight_sem >= mb_weight_sem_zdn, PT := waitTimeThrow);
		sem.run := FALSE;
		IF (ton2.Q = TRUE) THEN
			STEP := 3;
		END_IF;
	3 :	ftrig(CLK := skip.on_up);
		IF (ftrig.Q = TRUE) THEN
			temp := TRUE;
		END_IF;
		ton3(IN := temp, PT := waitTimeThrow);
		IF (mb_weight_sem > weight_sem_otkl - 1 AND ton3.Q = TRUE) THEN
			sem.open_cmd := run AND NOT mixerNoREADY;
		ELSE
			IF (ton3.Q = TRUE) THEN
				STEP := 0;
			END_IF;
			sem.open_cmd := FALSE;
		END_IF;
END_CASE;
IF (mb_weight_sem_zdn <= 0) THEN
	STEP := 0;
	run := FALSE;
END_IF;
END_PROGRAM

(* POU FTON, ST *)
FUNCTION_BLOCK FTON
VAR_INPUT
	IN : BOOL;
	PT : TIME;
END_VAR
VAR_OUTPUT
	Q : BOOL;
END_VAR
VAR
	ton1 : TON;
	ton2 : TON;
	temp : BOOL;
	trig1 : F_TRIG;
END_VAR
trig1(CLK := IN);
IF (trig1.Q = TRUE) THEN
	temp := TRUE;
END_IF;

ton1(IN := temp, PT := PT);
Q := ton1.Q;
ton2(IN := Q ,PT := T#2s);
IF (ton2.Q = TRUE) THEN
	temp := FALSE;
	ton1(IN := temp);
END_IF;
END_FUNCTION_BLOCK

(* POU RTON, ST *)
FUNCTION_BLOCK RTON
VAR_INPUT
	IN : BOOL;
	PT : TIME;
END_VAR
VAR_OUTPUT
	Q : BOOL;
END_VAR
VAR
	ton1 : TON;
	trig1 : R_TRIG;
	temp: BOOL;
END_VAR
trig1(CLK := IN);
IF (trig1.Q = TRUE) THEN
	temp := TRUE;
END_IF;
ton1(IN := temp, PT := PT);
Q := ton1.Q;
IF (ton1.Q = TRUE) THEN
	temp := FALSE;
END_IF;
END_FUNCTION_BLOCK

(* Visualisation jbi
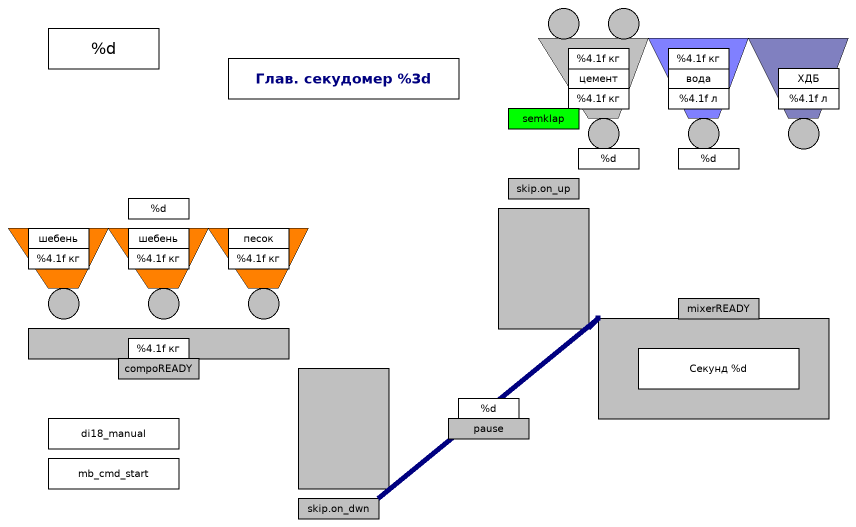
ellipse at (90,280)-(121,311): alarm colour if .do1_comp_1
ellipse at (190,280)-(221,311): alarm colour if .do2_comp_2
ellipse at (290,280)-(321,311): alarm colour if .do3_comp_3
rounded rectangle at (70,320)-(331,351): alarm colour if .con.run
rounded rectangle at (340,360)-(431,481): invisible if NOT .skip.on_down; alarm colour if .skip.cmd_up; angle 45
rounded rectangle at (540,200)-(631,321): invisible if NOT .skip.on_up; alarm colour if .skip.cmd_dwn; angle 45
polygon at (580,30)-(690,110): alarm colour if .sem.run
polygon at (690,30)-(790,110): alarm colour if ..do5_water_klap
ellipse at (630,110)-(661,141): alarm colour if .sem.open_cmd
ellipse at (730,110)-(761,141): alarm colour if .wtr.run
ellipse at (830,110)-(861,141): alarm colour if .plst.run
rounded rectangle at (640,310)-(871,411): alarm colour if .mixer.status; toggles .mdvv1_in.0
rounded rectangle at (270,50)-(501,91): text "Глав. секудомер %3d"; shows .GLOBT
rounded rectangle at (70,220)-(131,241): text "шебень"
rounded rectangle at (170,220)-(231,241): text "шебень"
rounded rectangle at (270,220)-(331,241): text "песок"
rounded rectangle at (170,330)-(231,351): text "%4.1f кг"; shows .mb_weight_sir; editable
rounded rectangle at (610,60)-(671,81): text "цемент"
rounded rectangle at (710,60)-(771,81): text "вода"
rounded rectangle at (820,60)-(881,81): text "ХДБ"
rounded rectangle at (610,80)-(671,101): text "%4.1f кг"; shows .mb_weight_sem; editable
rounded rectangle at (710,80)-(771,101): text "%4.1f л"; shows .mb_weight_water; editable
rounded rectangle at (820,80)-(881,101): text "%4.1f л"; shows .mb_weight_plast; editable
rounded rectangle at (550,170)-(621,191): text "skip.on_up"; alarm colour if .skip.on_up; toggles NOT .mdvv2_in.2
rounded rectangle at (340,490)-(421,511): text "skip.on_dwn"; alarm colour if .skip.on_down; toggles NOT .mdvv2_in.0
rectangle at (90,410)-(221,441): text "di18_manual"; alarm colour if .di18_sts_mnl; toggles .di18_sts_mnl
rectangle at (90,450)-(221,481): text "mb_cmd_start"; alarm colour if .mb_cmd_start; toggles .mb_cmd_start
rounded rectangle at (680,340)-(841,381): text "Секунд %d"; shows .cnt2.CV
rounded rectangle at (70,240)-(131,261): text "%4.1f кг"; shows .mb_weight_comp1_zdn; editable
rounded rectangle at (170,240)-(231,261): text "%4.1f кг"; shows .mb_weight_comp2_zdn; editable
rounded rectangle at (270,240)-(331,261): text "%4.1f кг"; shows .mb_weight_comp3_zdn; editable
rounded rectangle at (170,190)-(231,211): text "%d"; shows autoComponent.siklComp; editable
rounded rectangle at (90,20)-(201,61): text "%d"; shows .mb_sikl; editable
ellipse at (590,0)-(621,31): alarm colour if .mb_cmd_shnk1
ellipse at (650,0)-(681,31): alarm colour if .mb_cmd_shnk2
rounded rectangle at (610,40)-(671,61): text "%4.1f кг"; shows .mb_weight_sem_zdn; editable
rounded rectangle at (710,40)-(771,61): text "%4.1f кг"; shows .mb_weight_wtr_zdn; editable
rounded rectangle at (550,100)-(621,121): text "semklap"; alarm colour if .sem.klapCLOSE; toggles .sem.klapCLOSE
rounded rectangle at (620,140)-(681,161): text "%d"; shows autoSement.siklCement; editable
rounded rectangle at (500,390)-(561,411): text "%d"; shows autoSkip.siklSkip; editable
rounded rectangle at (720,290)-(801,311): text "mixerREADY"; alarm colour if .mixerREADY; toggles .mixerREADY
rounded rectangle at (160,350)-(241,371): text "compoREADY"; alarm colour if .componentsREADY; toggles .componentsREADY
rounded rectangle at (490,410)-(571,431): text "pause"; alarm colour if .mdvv2_in.10; toggles .mdvv2_in.10
rounded rectangle at (720,140)-(781,161): text "%d"; shows autoWater.siklWater; editable
5 more shapes without text or variables
*)
